FUNCTION_BLOCK LiftControl (* Basic Function Block Type *)
  (* Standard: 61499-2 *)
  (* Version 0.0, 1/14/2024, midxav, Template *)
  PACKAGE Main;
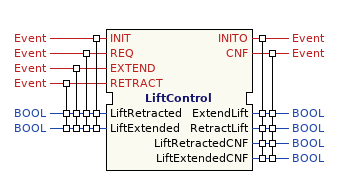
  EVENT_INPUT
    INIT WITH LiftRetracted, LiftExtended; (* Initialization Request *)
    REQ WITH LiftRetracted, LiftExtended; (* Normal Execution Request *)
    EXTEND WITH LiftRetracted, LiftExtended;
    RETRACT WITH LiftRetracted, LiftExtended;
  END_EVENT
  EVENT_OUTPUT
    INITO WITH ExtendLift, RetractLift, LiftRetractedCNF, LiftExtendedCNF; (* Initialization Confirm *)
    CNF WITH ExtendLift, RetractLift, LiftRetractedCNF, LiftExtendedCNF; (* Execution Confirmation *)
  END_EVENT
  VAR_INPUT
    LiftRetracted : BOOL; (* Input event qualifier *)
    LiftExtended : BOOL;
  END_VAR
  VAR_OUTPUT
    ExtendLift : BOOL; (* Output event qualifier *)
    RetractLift : BOOL;
    LiftRetractedCNF : BOOL;
    LiftExtendedCNF : BOOL;
  END_VAR
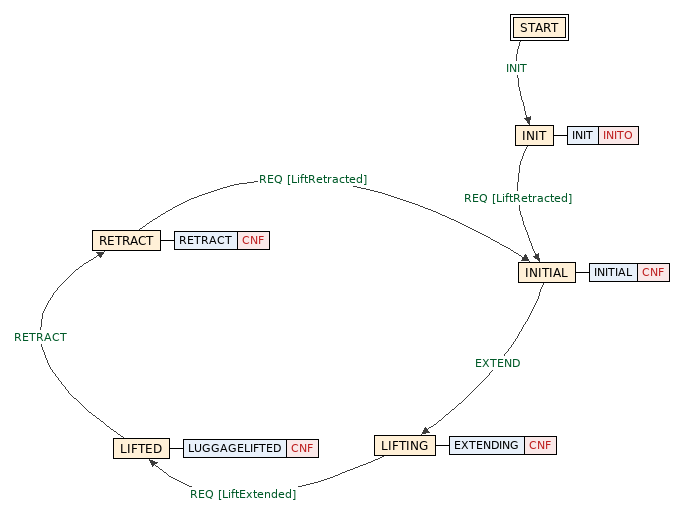
  EC_STATES
    START; (* Initial State *)
    INIT : INIT -> INITO; (* Initialization *)
    INITIAL : INITIAL -> CNF;
    LIFTING : EXTENDING -> CNF;
    LIFTED : LUGGAGELIFTED -> CNF;
    RETRACT : RETRACT -> CNF;
  END_STATES
  EC_TRANSITIONS
    START TO INIT := INIT;
    INIT TO INITIAL := REQ [LiftRetracted];
    INITIAL TO LIFTING := EXTEND;
    LIFTING TO LIFTED := REQ [LiftExtended];
    LIFTED TO RETRACT := RETRACT;
    RETRACT TO INITIAL := REQ [LiftRetracted];
  END_TRANSITIONS
  ALGORITHM INIT IN ST:
ExtendLift:= FALSE;
RetractLift:=TRUE;
LiftExtendedCNF := FALSE;
LiftRetractedCNF := FALSE;
  END_ALGORITHM
  ALGORITHM INITIAL IN ST:
RetractLift:=FALSE;
LiftExtendedCNF := FALSE;
LiftRetractedCNF := TRUE;
  END_ALGORITHM
  ALGORITHM EXTENDING IN ST:
ExtendLift:=TRUE;
LiftRetractedCNF := FALSE;
  END_ALGORITHM
  ALGORITHM LUGGAGELIFTED IN ST:
ExtendLift:=FALSE;
LiftExtendedCNF := TRUE;
  END_ALGORITHM
  ALGORITHM RETRACT IN ST:
RetractLift:=TRUE;
LiftExtendedCNF := FALSE;
  END_ALGORITHM
END_FUNCTION_BLOCK
